PROGRAM F25_CylindersCtrl
VAR
	aCylinderCtrl		:ARRAY[1..cMAX_CYLINDERS] OF  FB_Cylinder;

	bStationHomed		: BOOL;
	bSeqHomingRequest	: BOOL;
	bTestRelease			: BOOL;
END_VAR
VAR // added by the converter: edge detectors and wires of the graphical bodies
    _w1, _w2, _w3, _w4, _w5, _w6, _w7 : BOOL;
END_VAR

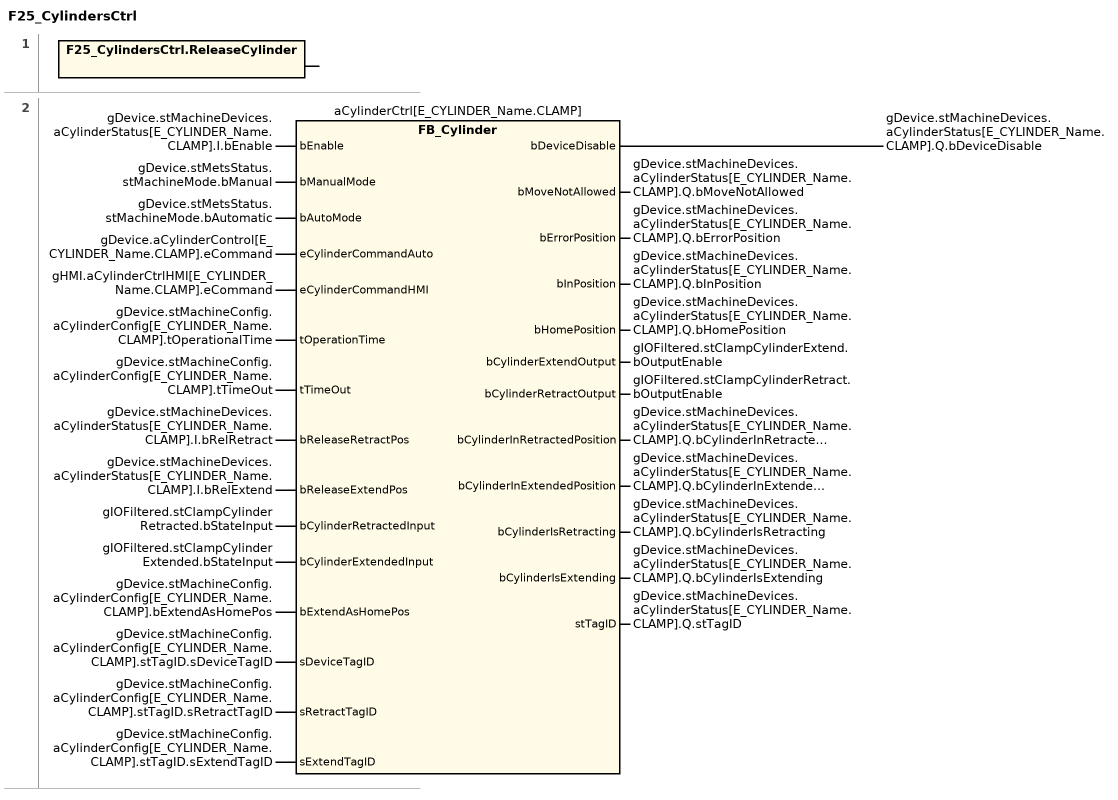
// NETWORK 1
F25_CylindersCtrl.ReleaseCylinder();

// NETWORK 2
aCylinderCtrl[E_CYLINDER_Name.CLAMP](
    bEnable := gDevice.stMachineDevices.aCylinderStatus[E_CYLINDER_Name.CLAMP].I.bEnable,
    bManualMode := gDevice.stMetsStatus.stMachineMode.bManual,
    bAutoMode := gDevice.stMetsStatus.stMachineMode.bAutomatic,
    eCylinderCommandAuto := gDevice.aCylinderControl[E_CYLINDER_Name.CLAMP].eCommand,
    eCylinderCommandHMI := gHMI.aCylinderCtrlHMI[E_CYLINDER_Name.CLAMP].eCommand,
    tOperationTime := gDevice.stMachineConfig.aCylinderConfig[E_CYLINDER_Name.CLAMP].tOperationalTime,
    tTimeOut := gDevice.stMachineConfig.aCylinderConfig[E_CYLINDER_Name.CLAMP].tTimeOut,
    bReleaseRetractPos := gDevice.stMachineDevices.aCylinderStatus[E_CYLINDER_Name.CLAMP].I.bRelRetract,
    bReleaseExtendPos := gDevice.stMachineDevices.aCylinderStatus[E_CYLINDER_Name.CLAMP].I.bRelExtend,
    bCylinderRetractedInput := gIOFiltered.stClampCylinderRetracted.bStateInput,
    bCylinderExtendedInput := gIOFiltered.stClampCylinderExtended.bStateInput,
    bExtendAsHomePos := gDevice.stMachineConfig.aCylinderConfig[E_CYLINDER_Name.CLAMP].bExtendAsHomePos,
    sDeviceTagID := gDevice.stMachineConfig.aCylinderConfig[E_CYLINDER_Name.CLAMP].stTagID.sDeviceTagID,
    sRetractTagID := gDevice.stMachineConfig.aCylinderConfig[E_CYLINDER_Name.CLAMP].stTagID.sRetractTagID,
    sExtendTagID := gDevice.stMachineConfig.aCylinderConfig[E_CYLINDER_Name.CLAMP].stTagID.sExtendTagID,
    bMoveNotAllowed => gDevice.stMachineDevices.aCylinderStatus[E_CYLINDER_Name.CLAMP].Q.bMoveNotAllowed,
    bErrorPosition => gDevice.stMachineDevices.aCylinderStatus[E_CYLINDER_Name.CLAMP].Q.bErrorPosition,
    bInPosition => gDevice.stMachineDevices.aCylinderStatus[E_CYLINDER_Name.CLAMP].Q.bInPosition,
    bHomePosition => gDevice.stMachineDevices.aCylinderStatus[E_CYLINDER_Name.CLAMP].Q.bHomePosition,
    bCylinderExtendOutput => gIOFiltered.stClampCylinderExtend.bOutputEnable,
    bCylinderRetractOutput => gIOFiltered.stClampCylinderRetract.bOutputEnable,
    bCylinderInRetractedPosition => gDevice.stMachineDevices.aCylinderStatus[E_CYLINDER_Name.CLAMP].Q.bCylinderInRetractedPosition,
    bCylinderInExtendedPosition => gDevice.stMachineDevices.aCylinderStatus[E_CYLINDER_Name.CLAMP].Q.bCylinderInExtendedPosition,
    bCylinderIsRetracting => gDevice.stMachineDevices.aCylinderStatus[E_CYLINDER_Name.CLAMP].Q.bCylinderIsRetracting,
    bCylinderIsExtending => gDevice.stMachineDevices.aCylinderStatus[E_CYLINDER_Name.CLAMP].Q.bCylinderIsExtending,
    stTagID => gDevice.stMachineDevices.aCylinderStatus[E_CYLINDER_Name.CLAMP].Q.stTagID); // FB_Cylinder
gDevice.stMachineDevices.aCylinderStatus[E_CYLINDER_Name.CLAMP].Q.bDeviceDisable := aCylinderCtrl[E_CYLINDER_Name.CLAMP].bDeviceDisable;

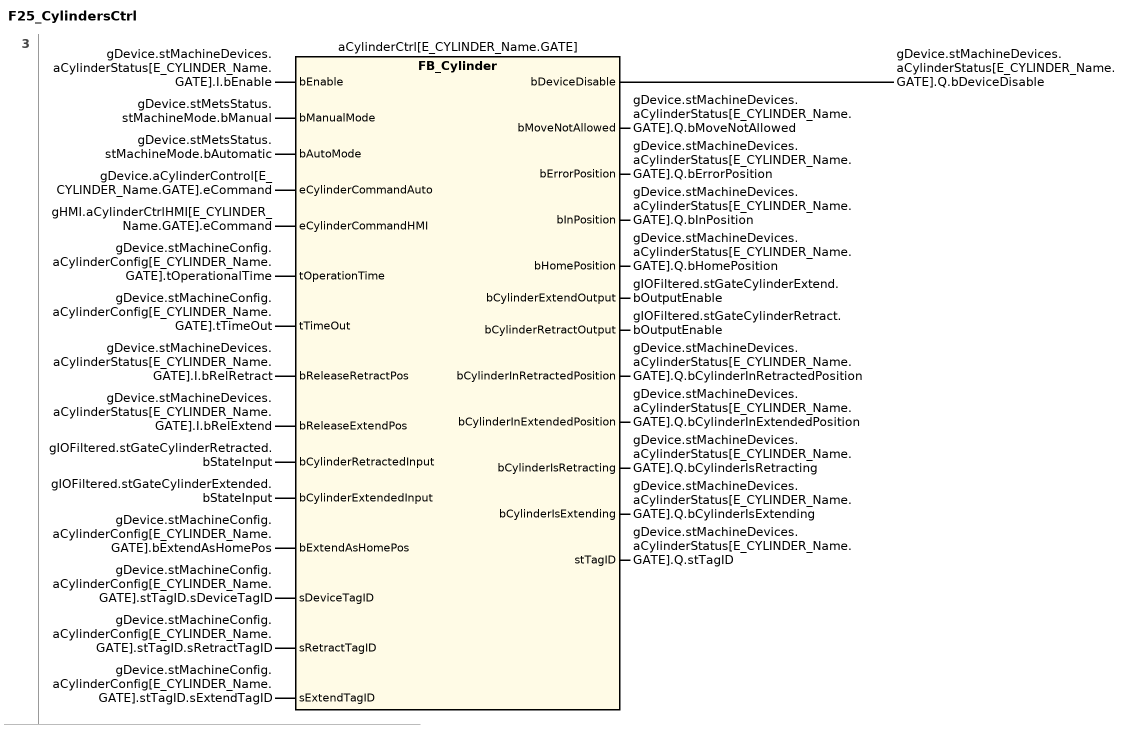
// NETWORK 3
aCylinderCtrl[E_CYLINDER_Name.GATE](
    bEnable := gDevice.stMachineDevices.aCylinderStatus[E_CYLINDER_Name.GATE].I.bEnable,
    bManualMode := gDevice.stMetsStatus.stMachineMode.bManual,
    bAutoMode := gDevice.stMetsStatus.stMachineMode.bAutomatic,
    eCylinderCommandAuto := gDevice.aCylinderControl[E_CYLINDER_Name.GATE].eCommand,
    eCylinderCommandHMI := gHMI.aCylinderCtrlHMI[E_CYLINDER_Name.GATE].eCommand,
    tOperationTime := gDevice.stMachineConfig.aCylinderConfig[E_CYLINDER_Name.GATE].tOperationalTime,
    tTimeOut := gDevice.stMachineConfig.aCylinderConfig[E_CYLINDER_Name.GATE].tTimeOut,
    bReleaseRetractPos := gDevice.stMachineDevices.aCylinderStatus[E_CYLINDER_Name.GATE].I.bRelRetract,
    bReleaseExtendPos := gDevice.stMachineDevices.aCylinderStatus[E_CYLINDER_Name.GATE].I.bRelExtend,
    bCylinderRetractedInput := gIOFiltered.stGateCylinderRetracted.bStateInput,
    bCylinderExtendedInput := gIOFiltered.stGateCylinderExtended.bStateInput,
    bExtendAsHomePos := gDevice.stMachineConfig.aCylinderConfig[E_CYLINDER_Name.GATE].bExtendAsHomePos,
    sDeviceTagID := gDevice.stMachineConfig.aCylinderConfig[E_CYLINDER_Name.GATE].stTagID.sDeviceTagID,
    sRetractTagID := gDevice.stMachineConfig.aCylinderConfig[E_CYLINDER_Name.GATE].stTagID.sRetractTagID,
    sExtendTagID := gDevice.stMachineConfig.aCylinderConfig[E_CYLINDER_Name.GATE].stTagID.sExtendTagID,
    bMoveNotAllowed => gDevice.stMachineDevices.aCylinderStatus[E_CYLINDER_Name.GATE].Q.bMoveNotAllowed,
    bErrorPosition => gDevice.stMachineDevices.aCylinderStatus[E_CYLINDER_Name.GATE].Q.bErrorPosition,
    bInPosition => gDevice.stMachineDevices.aCylinderStatus[E_CYLINDER_Name.GATE].Q.bInPosition,
    bHomePosition => gDevice.stMachineDevices.aCylinderStatus[E_CYLINDER_Name.GATE].Q.bHomePosition,
    bCylinderExtendOutput => gIOFiltered.stGateCylinderExtend.bOutputEnable,
    bCylinderRetractOutput => gIOFiltered.stGateCylinderRetract.bOutputEnable,
    bCylinderInRetractedPosition => gDevice.stMachineDevices.aCylinderStatus[E_CYLINDER_Name.GATE].Q.bCylinderInRetractedPosition,
    bCylinderInExtendedPosition => gDevice.stMachineDevices.aCylinderStatus[E_CYLINDER_Name.GATE].Q.bCylinderInExtendedPosition,
    bCylinderIsRetracting => gDevice.stMachineDevices.aCylinderStatus[E_CYLINDER_Name.GATE].Q.bCylinderIsRetracting,
    bCylinderIsExtending => gDevice.stMachineDevices.aCylinderStatus[E_CYLINDER_Name.GATE].Q.bCylinderIsExtending,
    stTagID => gDevice.stMachineDevices.aCylinderStatus[E_CYLINDER_Name.GATE].Q.stTagID); // FB_Cylinder
gDevice.stMachineDevices.aCylinderStatus[E_CYLINDER_Name.GATE].Q.bDeviceDisable := aCylinderCtrl[E_CYLINDER_Name.GATE].bDeviceDisable;

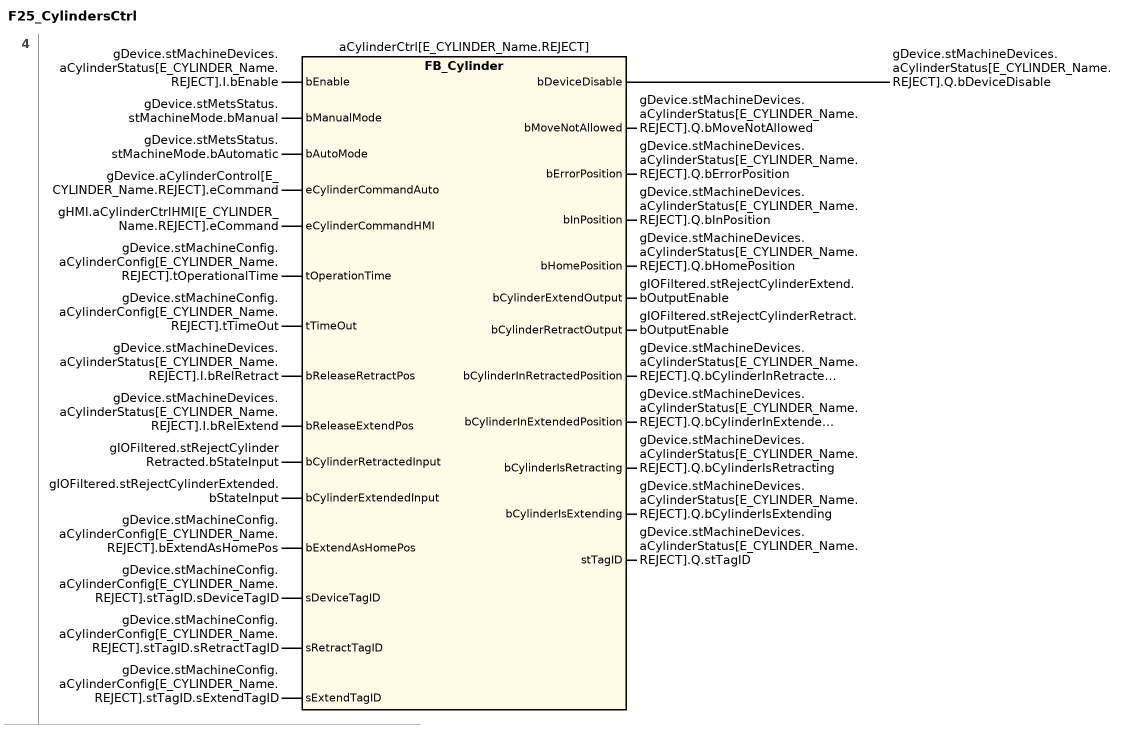
// NETWORK 4
aCylinderCtrl[E_CYLINDER_Name.REJECT](
    bEnable := gDevice.stMachineDevices.aCylinderStatus[E_CYLINDER_Name.REJECT].I.bEnable,
    bManualMode := gDevice.stMetsStatus.stMachineMode.bManual,
    bAutoMode := gDevice.stMetsStatus.stMachineMode.bAutomatic,
    eCylinderCommandAuto := gDevice.aCylinderControl[E_CYLINDER_Name.REJECT].eCommand,
    eCylinderCommandHMI := gHMI.aCylinderCtrlHMI[E_CYLINDER_Name.REJECT].eCommand,
    tOperationTime := gDevice.stMachineConfig.aCylinderConfig[E_CYLINDER_Name.REJECT].tOperationalTime,
    tTimeOut := gDevice.stMachineConfig.aCylinderConfig[E_CYLINDER_Name.REJECT].tTimeOut,
    bReleaseRetractPos := gDevice.stMachineDevices.aCylinderStatus[E_CYLINDER_Name.REJECT].I.bRelRetract,
    bReleaseExtendPos := gDevice.stMachineDevices.aCylinderStatus[E_CYLINDER_Name.REJECT].I.bRelExtend,
    bCylinderRetractedInput := gIOFiltered.stRejectCylinderRetracted.bStateInput,
    bCylinderExtendedInput := gIOFiltered.stRejectCylinderExtended.bStateInput,
    bExtendAsHomePos := gDevice.stMachineConfig.aCylinderConfig[E_CYLINDER_Name.REJECT].bExtendAsHomePos,
    sDeviceTagID := gDevice.stMachineConfig.aCylinderConfig[E_CYLINDER_Name.REJECT].stTagID.sDeviceTagID,
    sRetractTagID := gDevice.stMachineConfig.aCylinderConfig[E_CYLINDER_Name.REJECT].stTagID.sRetractTagID,
    sExtendTagID := gDevice.stMachineConfig.aCylinderConfig[E_CYLINDER_Name.REJECT].stTagID.sExtendTagID,
    bMoveNotAllowed => gDevice.stMachineDevices.aCylinderStatus[E_CYLINDER_Name.REJECT].Q.bMoveNotAllowed,
    bErrorPosition => gDevice.stMachineDevices.aCylinderStatus[E_CYLINDER_Name.REJECT].Q.bErrorPosition,
    bInPosition => gDevice.stMachineDevices.aCylinderStatus[E_CYLINDER_Name.REJECT].Q.bInPosition,
    bHomePosition => gDevice.stMachineDevices.aCylinderStatus[E_CYLINDER_Name.REJECT].Q.bHomePosition,
    bCylinderExtendOutput => gIOFiltered.stRejectCylinderExtend.bOutputEnable,
    bCylinderRetractOutput => gIOFiltered.stRejectCylinderRetract.bOutputEnable,
    bCylinderInRetractedPosition => gDevice.stMachineDevices.aCylinderStatus[E_CYLINDER_Name.REJECT].Q.bCylinderInRetractedPosition,
    bCylinderInExtendedPosition => gDevice.stMachineDevices.aCylinderStatus[E_CYLINDER_Name.REJECT].Q.bCylinderInExtendedPosition,
    bCylinderIsRetracting => gDevice.stMachineDevices.aCylinderStatus[E_CYLINDER_Name.REJECT].Q.bCylinderIsRetracting,
    bCylinderIsExtending => gDevice.stMachineDevices.aCylinderStatus[E_CYLINDER_Name.REJECT].Q.bCylinderIsExtending,
    stTagID => gDevice.stMachineDevices.aCylinderStatus[E_CYLINDER_Name.REJECT].Q.stTagID); // FB_Cylinder
gDevice.stMachineDevices.aCylinderStatus[E_CYLINDER_Name.REJECT].Q.bDeviceDisable := aCylinderCtrl[E_CYLINDER_Name.REJECT].bDeviceDisable;

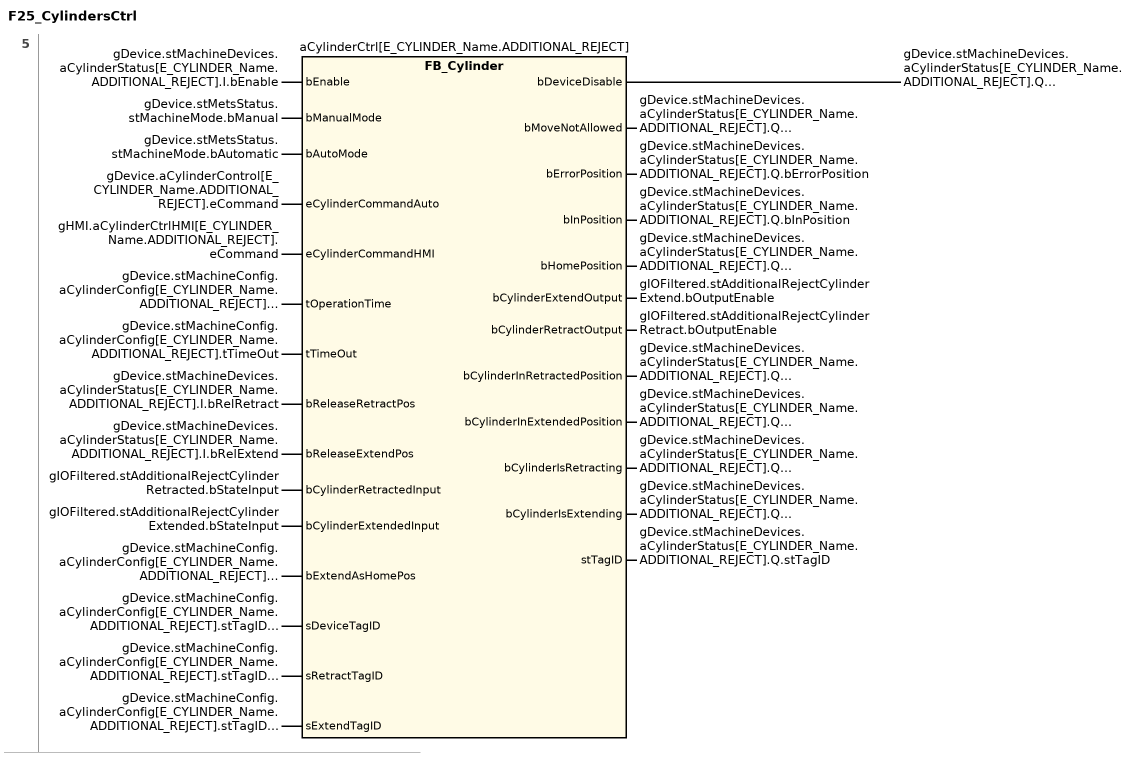
// NETWORK 5
aCylinderCtrl[E_CYLINDER_Name.ADDITIONAL_REJECT](
    bEnable := gDevice.stMachineDevices.aCylinderStatus[E_CYLINDER_Name.ADDITIONAL_REJECT].I.bEnable,
    bManualMode := gDevice.stMetsStatus.stMachineMode.bManual,
    bAutoMode := gDevice.stMetsStatus.stMachineMode.bAutomatic,
    eCylinderCommandAuto := gDevice.aCylinderControl[E_CYLINDER_Name.ADDITIONAL_REJECT].eCommand,
    eCylinderCommandHMI := gHMI.aCylinderCtrlHMI[E_CYLINDER_Name.ADDITIONAL_REJECT].eCommand,
    tOperationTime := gDevice.stMachineConfig.aCylinderConfig[E_CYLINDER_Name.ADDITIONAL_REJECT].tOperationalTime,
    tTimeOut := gDevice.stMachineConfig.aCylinderConfig[E_CYLINDER_Name.ADDITIONAL_REJECT].tTimeOut,
    bReleaseRetractPos := gDevice.stMachineDevices.aCylinderStatus[E_CYLINDER_Name.ADDITIONAL_REJECT].I.bRelRetract,
    bReleaseExtendPos := gDevice.stMachineDevices.aCylinderStatus[E_CYLINDER_Name.ADDITIONAL_REJECT].I.bRelExtend,
    bCylinderRetractedInput := gIOFiltered.stAdditionalRejectCylinderRetracted.bStateInput,
    bCylinderExtendedInput := gIOFiltered.stAdditionalRejectCylinderExtended.bStateInput,
    bExtendAsHomePos := gDevice.stMachineConfig.aCylinderConfig[E_CYLINDER_Name.ADDITIONAL_REJECT].bExtendAsHomePos,
    sDeviceTagID := gDevice.stMachineConfig.aCylinderConfig[E_CYLINDER_Name.ADDITIONAL_REJECT].stTagID.sDeviceTagID,
    sRetractTagID := gDevice.stMachineConfig.aCylinderConfig[E_CYLINDER_Name.ADDITIONAL_REJECT].stTagID.sRetractTagID,
    sExtendTagID := gDevice.stMachineConfig.aCylinderConfig[E_CYLINDER_Name.ADDITIONAL_REJECT].stTagID.sExtendTagID,
    bMoveNotAllowed => gDevice.stMachineDevices.aCylinderStatus[E_CYLINDER_Name.ADDITIONAL_REJECT].Q.bMoveNotAllowed,
    bErrorPosition => gDevice.stMachineDevices.aCylinderStatus[E_CYLINDER_Name.ADDITIONAL_REJECT].Q.bErrorPosition,
    bInPosition => gDevice.stMachineDevices.aCylinderStatus[E_CYLINDER_Name.ADDITIONAL_REJECT].Q.bInPosition,
    bHomePosition => gDevice.stMachineDevices.aCylinderStatus[E_CYLINDER_Name.ADDITIONAL_REJECT].Q.bHomePosition,
    bCylinderExtendOutput => gIOFiltered.stAdditionalRejectCylinderExtend.bOutputEnable,
    bCylinderRetractOutput => gIOFiltered.stAdditionalRejectCylinderRetract.bOutputEnable,
    bCylinderInRetractedPosition => gDevice.stMachineDevices.aCylinderStatus[E_CYLINDER_Name.ADDITIONAL_REJECT].Q.bCylinderInRetractedPosition,
    bCylinderInExtendedPosition => gDevice.stMachineDevices.aCylinderStatus[E_CYLINDER_Name.ADDITIONAL_REJECT].Q.bCylinderInExtendedPosition,
    bCylinderIsRetracting => gDevice.stMachineDevices.aCylinderStatus[E_CYLINDER_Name.ADDITIONAL_REJECT].Q.bCylinderIsRetracting,
    bCylinderIsExtending => gDevice.stMachineDevices.aCylinderStatus[E_CYLINDER_Name.ADDITIONAL_REJECT].Q.bCylinderIsExtending,
    stTagID => gDevice.stMachineDevices.aCylinderStatus[E_CYLINDER_Name.ADDITIONAL_REJECT].Q.stTagID); // FB_Cylinder
gDevice.stMachineDevices.aCylinderStatus[E_CYLINDER_Name.ADDITIONAL_REJECT].Q.bDeviceDisable := aCylinderCtrl[E_CYLINDER_Name.ADDITIONAL_REJECT].bDeviceDisable;

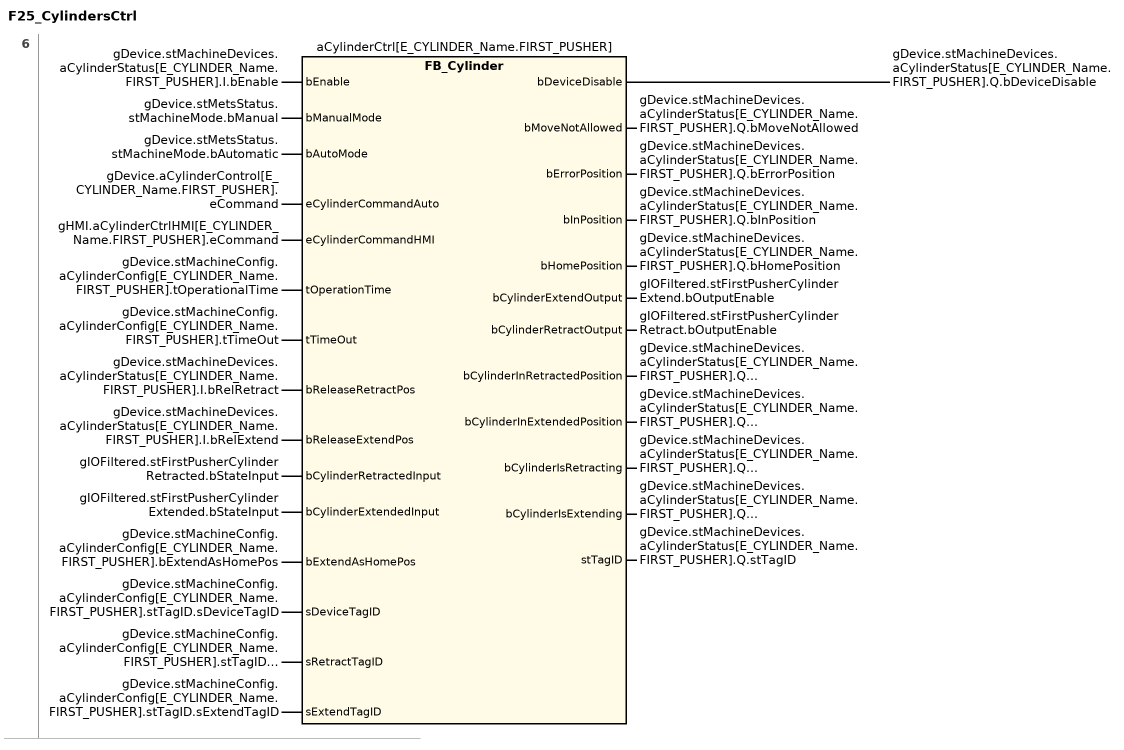
// NETWORK 6
aCylinderCtrl[E_CYLINDER_Name.FIRST_PUSHER](
    bEnable := gDevice.stMachineDevices.aCylinderStatus[E_CYLINDER_Name.FIRST_PUSHER].I.bEnable,
    bManualMode := gDevice.stMetsStatus.stMachineMode.bManual,
    bAutoMode := gDevice.stMetsStatus.stMachineMode.bAutomatic,
    eCylinderCommandAuto := gDevice.aCylinderControl[E_CYLINDER_Name.FIRST_PUSHER].eCommand,
    eCylinderCommandHMI := gHMI.aCylinderCtrlHMI[E_CYLINDER_Name.FIRST_PUSHER].eCommand,
    tOperationTime := gDevice.stMachineConfig.aCylinderConfig[E_CYLINDER_Name.FIRST_PUSHER].tOperationalTime,
    tTimeOut := gDevice.stMachineConfig.aCylinderConfig[E_CYLINDER_Name.FIRST_PUSHER].tTimeOut,
    bReleaseRetractPos := gDevice.stMachineDevices.aCylinderStatus[E_CYLINDER_Name.FIRST_PUSHER].I.bRelRetract,
    bReleaseExtendPos := gDevice.stMachineDevices.aCylinderStatus[E_CYLINDER_Name.FIRST_PUSHER].I.bRelExtend,
    bCylinderRetractedInput := gIOFiltered.stFirstPusherCylinderRetracted.bStateInput,
    bCylinderExtendedInput := gIOFiltered.stFirstPusherCylinderExtended.bStateInput,
    bExtendAsHomePos := gDevice.stMachineConfig.aCylinderConfig[E_CYLINDER_Name.FIRST_PUSHER].bExtendAsHomePos,
    sDeviceTagID := gDevice.stMachineConfig.aCylinderConfig[E_CYLINDER_Name.FIRST_PUSHER].stTagID.sDeviceTagID,
    sRetractTagID := gDevice.stMachineConfig.aCylinderConfig[E_CYLINDER_Name.FIRST_PUSHER].stTagID.sRetractTagID,
    sExtendTagID := gDevice.stMachineConfig.aCylinderConfig[E_CYLINDER_Name.FIRST_PUSHER].stTagID.sExtendTagID,
    bMoveNotAllowed => gDevice.stMachineDevices.aCylinderStatus[E_CYLINDER_Name.FIRST_PUSHER].Q.bMoveNotAllowed,
    bErrorPosition => gDevice.stMachineDevices.aCylinderStatus[E_CYLINDER_Name.FIRST_PUSHER].Q.bErrorPosition,
    bInPosition => gDevice.stMachineDevices.aCylinderStatus[E_CYLINDER_Name.FIRST_PUSHER].Q.bInPosition,
    bHomePosition => gDevice.stMachineDevices.aCylinderStatus[E_CYLINDER_Name.FIRST_PUSHER].Q.bHomePosition,
    bCylinderExtendOutput => gIOFiltered.stFirstPusherCylinderExtend.bOutputEnable,
    bCylinderRetractOutput => gIOFiltered.stFirstPusherCylinderRetract.bOutputEnable,
    bCylinderInRetractedPosition => gDevice.stMachineDevices.aCylinderStatus[E_CYLINDER_Name.FIRST_PUSHER].Q.bCylinderInRetractedPosition,
    bCylinderInExtendedPosition => gDevice.stMachineDevices.aCylinderStatus[E_CYLINDER_Name.FIRST_PUSHER].Q.bCylinderInExtendedPosition,
    bCylinderIsRetracting => gDevice.stMachineDevices.aCylinderStatus[E_CYLINDER_Name.FIRST_PUSHER].Q.bCylinderIsRetracting,
    bCylinderIsExtending => gDevice.stMachineDevices.aCylinderStatus[E_CYLINDER_Name.FIRST_PUSHER].Q.bCylinderIsExtending,
    stTagID => gDevice.stMachineDevices.aCylinderStatus[E_CYLINDER_Name.FIRST_PUSHER].Q.stTagID); // FB_Cylinder
gDevice.stMachineDevices.aCylinderStatus[E_CYLINDER_Name.FIRST_PUSHER].Q.bDeviceDisable := aCylinderCtrl[E_CYLINDER_Name.FIRST_PUSHER].bDeviceDisable;

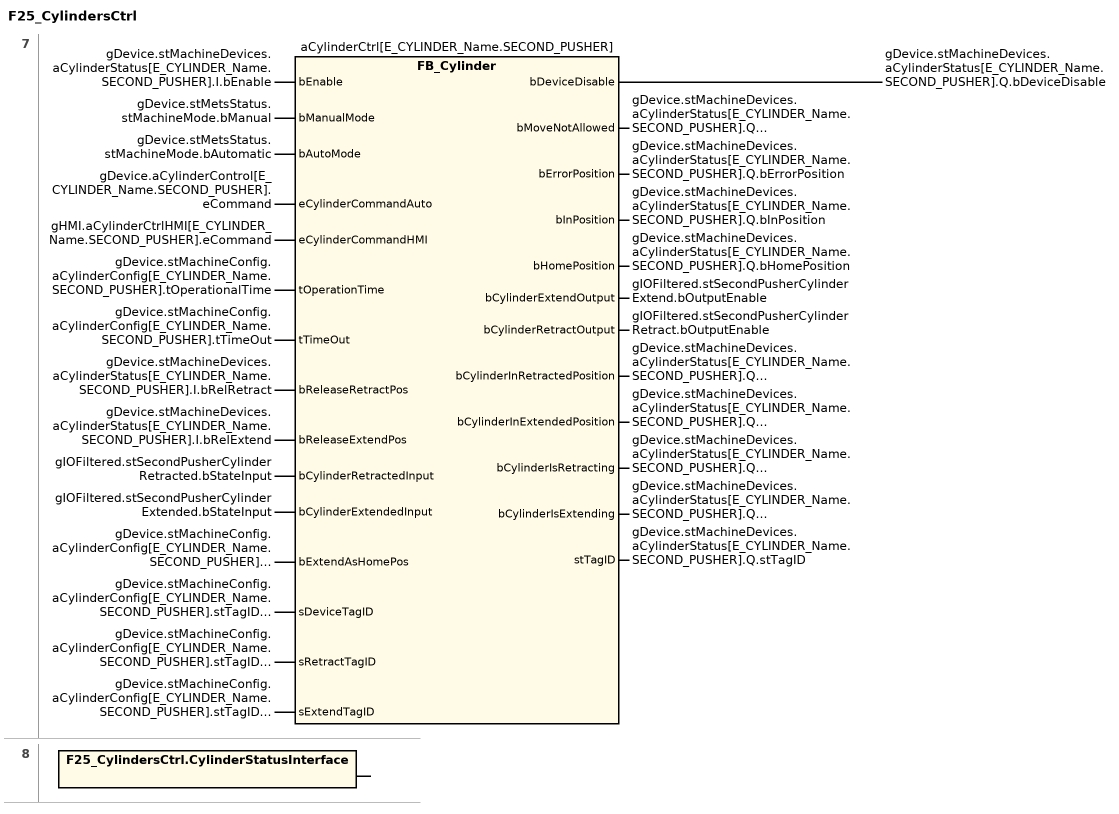
// NETWORK 7
aCylinderCtrl[E_CYLINDER_Name.SECOND_PUSHER](
    bEnable := gDevice.stMachineDevices.aCylinderStatus[E_CYLINDER_Name.SECOND_PUSHER].I.bEnable,
    bManualMode := gDevice.stMetsStatus.stMachineMode.bManual,
    bAutoMode := gDevice.stMetsStatus.stMachineMode.bAutomatic,
    eCylinderCommandAuto := gDevice.aCylinderControl[E_CYLINDER_Name.SECOND_PUSHER].eCommand,
    eCylinderCommandHMI := gHMI.aCylinderCtrlHMI[E_CYLINDER_Name.SECOND_PUSHER].eCommand,
    tOperationTime := gDevice.stMachineConfig.aCylinderConfig[E_CYLINDER_Name.SECOND_PUSHER].tOperationalTime,
    tTimeOut := gDevice.stMachineConfig.aCylinderConfig[E_CYLINDER_Name.SECOND_PUSHER].tTimeOut,
    bReleaseRetractPos := gDevice.stMachineDevices.aCylinderStatus[E_CYLINDER_Name.SECOND_PUSHER].I.bRelRetract,
    bReleaseExtendPos := gDevice.stMachineDevices.aCylinderStatus[E_CYLINDER_Name.SECOND_PUSHER].I.bRelExtend,
    bCylinderRetractedInput := gIOFiltered.stSecondPusherCylinderRetracted.bStateInput,
    bCylinderExtendedInput := gIOFiltered.stSecondPusherCylinderExtended.bStateInput,
    bExtendAsHomePos := gDevice.stMachineConfig.aCylinderConfig[E_CYLINDER_Name.SECOND_PUSHER].bExtendAsHomePos,
    sDeviceTagID := gDevice.stMachineConfig.aCylinderConfig[E_CYLINDER_Name.SECOND_PUSHER].stTagID.sDeviceTagID,
    sRetractTagID := gDevice.stMachineConfig.aCylinderConfig[E_CYLINDER_Name.SECOND_PUSHER].stTagID.sRetractTagID,
    sExtendTagID := gDevice.stMachineConfig.aCylinderConfig[E_CYLINDER_Name.SECOND_PUSHER].stTagID.sExtendTagID,
    bMoveNotAllowed => gDevice.stMachineDevices.aCylinderStatus[E_CYLINDER_Name.SECOND_PUSHER].Q.bMoveNotAllowed,
    bErrorPosition => gDevice.stMachineDevices.aCylinderStatus[E_CYLINDER_Name.SECOND_PUSHER].Q.bErrorPosition,
    bInPosition => gDevice.stMachineDevices.aCylinderStatus[E_CYLINDER_Name.SECOND_PUSHER].Q.bInPosition,
    bHomePosition => gDevice.stMachineDevices.aCylinderStatus[E_CYLINDER_Name.SECOND_PUSHER].Q.bHomePosition,
    bCylinderExtendOutput => gIOFiltered.stSecondPusherCylinderExtend.bOutputEnable,
    bCylinderRetractOutput => gIOFiltered.stSecondPusherCylinderRetract.bOutputEnable,
    bCylinderInRetractedPosition => gDevice.stMachineDevices.aCylinderStatus[E_CYLINDER_Name.SECOND_PUSHER].Q.bCylinderInRetractedPosition,
    bCylinderInExtendedPosition => gDevice.stMachineDevices.aCylinderStatus[E_CYLINDER_Name.SECOND_PUSHER].Q.bCylinderInExtendedPosition,
    bCylinderIsRetracting => gDevice.stMachineDevices.aCylinderStatus[E_CYLINDER_Name.SECOND_PUSHER].Q.bCylinderIsRetracting,
    bCylinderIsExtending => gDevice.stMachineDevices.aCylinderStatus[E_CYLINDER_Name.SECOND_PUSHER].Q.bCylinderIsExtending,
    stTagID => gDevice.stMachineDevices.aCylinderStatus[E_CYLINDER_Name.SECOND_PUSHER].Q.stTagID); // FB_Cylinder
gDevice.stMachineDevices.aCylinderStatus[E_CYLINDER_Name.SECOND_PUSHER].Q.bDeviceDisable := aCylinderCtrl[E_CYLINDER_Name.SECOND_PUSHER].bDeviceDisable;

// NETWORK 8
F25_CylindersCtrl.CylinderStatusInterface();

ACTION CylinderStatusInterface:
MEMMOVE(ADR(gHMI.aCylinderStatusHMI[E_CYLINDER_Name.CLAMP]), ADR(gDevice.stMachineDevices.aCylinderStatus[E_CYLINDER_Name.CLAMP].Q),SIZEOF( gDevice.stMachineDevices.aCylinderStatus[E_CYLINDER_Name.CLAMP].Q));
MEMMOVE(ADR(gHMI.aCylinderStatusHMI[E_CYLINDER_Name.GATE]), ADR(gDevice.stMachineDevices.aCylinderStatus[E_CYLINDER_Name.GATE].Q),SIZEOF( gDevice.stMachineDevices.aCylinderStatus[E_CYLINDER_Name.GATE].Q));
MEMMOVE(ADR(gHMI.aCylinderStatusHMI[E_CYLINDER_Name.REJECT]), ADR(gDevice.stMachineDevices.aCylinderStatus[E_CYLINDER_Name.REJECT].Q),SIZEOF( gDevice.stMachineDevices.aCylinderStatus[E_CYLINDER_Name.REJECT].Q));
MEMMOVE(ADR(gHMI.aCylinderStatusHMI[E_CYLINDER_Name.ADDITIONAL_REJECT]), ADR(gDevice.stMachineDevices.aCylinderStatus[E_CYLINDER_Name.ADDITIONAL_REJECT].Q),SIZEOF( gDevice.stMachineDevices.aCylinderStatus[E_CYLINDER_Name.ADDITIONAL_REJECT].Q));
MEMMOVE(ADR(gHMI.aCylinderStatusHMI[E_CYLINDER_Name.FIRST_PUSHER]), ADR(gDevice.stMachineDevices.aCylinderStatus[E_CYLINDER_Name.FIRST_PUSHER].Q),SIZEOF( gDevice.stMachineDevices.aCylinderStatus[E_CYLINDER_Name.FIRST_PUSHER].Q));
MEMMOVE(ADR(gHMI.aCylinderStatusHMI[E_CYLINDER_Name.SECOND_PUSHER]), ADR(gDevice.stMachineDevices.aCylinderStatus[E_CYLINDER_Name.SECOND_PUSHER].Q),SIZEOF( gDevice.stMachineDevices.aCylinderStatus[E_CYLINDER_Name.SECOND_PUSHER].Q));
END_ACTION

ACTION ReleaseCylinder:
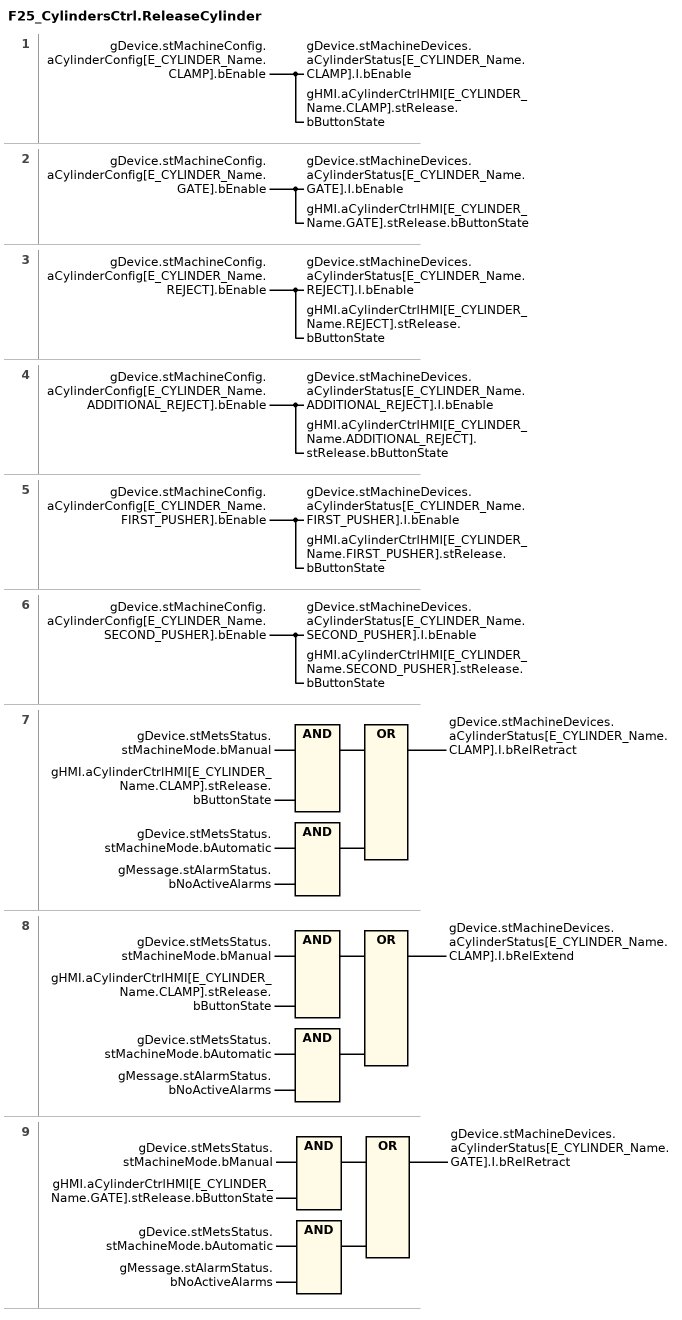
// NETWORK 1
_w1 := gDevice.stMachineConfig.aCylinderConfig[E_CYLINDER_Name.CLAMP].bEnable;
gDevice.stMachineDevices.aCylinderStatus[E_CYLINDER_Name.CLAMP].I.bEnable := _w1;
gHMI.aCylinderCtrlHMI[E_CYLINDER_Name.CLAMP].stRelease.bButtonState := _w1;

// NETWORK 2
_w2 := gDevice.stMachineConfig.aCylinderConfig[E_CYLINDER_Name.GATE].bEnable;
gDevice.stMachineDevices.aCylinderStatus[E_CYLINDER_Name.GATE].I.bEnable := _w2;
gHMI.aCylinderCtrlHMI[E_CYLINDER_Name.GATE].stRelease.bButtonState := _w2;

// NETWORK 3
_w3 := gDevice.stMachineConfig.aCylinderConfig[E_CYLINDER_Name.REJECT].bEnable;
gDevice.stMachineDevices.aCylinderStatus[E_CYLINDER_Name.REJECT].I.bEnable := _w3;
gHMI.aCylinderCtrlHMI[E_CYLINDER_Name.REJECT].stRelease.bButtonState := _w3;

// NETWORK 4
_w4 := gDevice.stMachineConfig.aCylinderConfig[E_CYLINDER_Name.ADDITIONAL_REJECT].bEnable;
gDevice.stMachineDevices.aCylinderStatus[E_CYLINDER_Name.ADDITIONAL_REJECT].I.bEnable := _w4;
gHMI.aCylinderCtrlHMI[E_CYLINDER_Name.ADDITIONAL_REJECT].stRelease.bButtonState := _w4;

// NETWORK 5
_w5 := gDevice.stMachineConfig.aCylinderConfig[E_CYLINDER_Name.FIRST_PUSHER].bEnable;
gDevice.stMachineDevices.aCylinderStatus[E_CYLINDER_Name.FIRST_PUSHER].I.bEnable := _w5;
gHMI.aCylinderCtrlHMI[E_CYLINDER_Name.FIRST_PUSHER].stRelease.bButtonState := _w5;

// NETWORK 6
_w6 := gDevice.stMachineConfig.aCylinderConfig[E_CYLINDER_Name.SECOND_PUSHER].bEnable;
gDevice.stMachineDevices.aCylinderStatus[E_CYLINDER_Name.SECOND_PUSHER].I.bEnable := _w6;
gHMI.aCylinderCtrlHMI[E_CYLINDER_Name.SECOND_PUSHER].stRelease.bButtonState := _w6;

// NETWORK 7
gDevice.stMachineDevices.aCylinderStatus[E_CYLINDER_Name.CLAMP].I.bRelRetract := gDevice.stMetsStatus.stMachineMode.bManual AND gHMI.aCylinderCtrlHMI[E_CYLINDER_Name.CLAMP].stRelease.bButtonState OR gDevice.stMetsStatus.stMachineMode.bAutomatic AND gMessage.stAlarmStatus.bNoActiveAlarms;

// NETWORK 8
gDevice.stMachineDevices.aCylinderStatus[E_CYLINDER_Name.CLAMP].I.bRelExtend := gDevice.stMetsStatus.stMachineMode.bManual AND gHMI.aCylinderCtrlHMI[E_CYLINDER_Name.CLAMP].stRelease.bButtonState OR gDevice.stMetsStatus.stMachineMode.bAutomatic AND gMessage.stAlarmStatus.bNoActiveAlarms;

// NETWORK 9
gDevice.stMachineDevices.aCylinderStatus[E_CYLINDER_Name.GATE].I.bRelRetract := gDevice.stMetsStatus.stMachineMode.bManual AND gHMI.aCylinderCtrlHMI[E_CYLINDER_Name.GATE].stRelease.bButtonState OR gDevice.stMetsStatus.stMachineMode.bAutomatic AND gMessage.stAlarmStatus.bNoActiveAlarms;

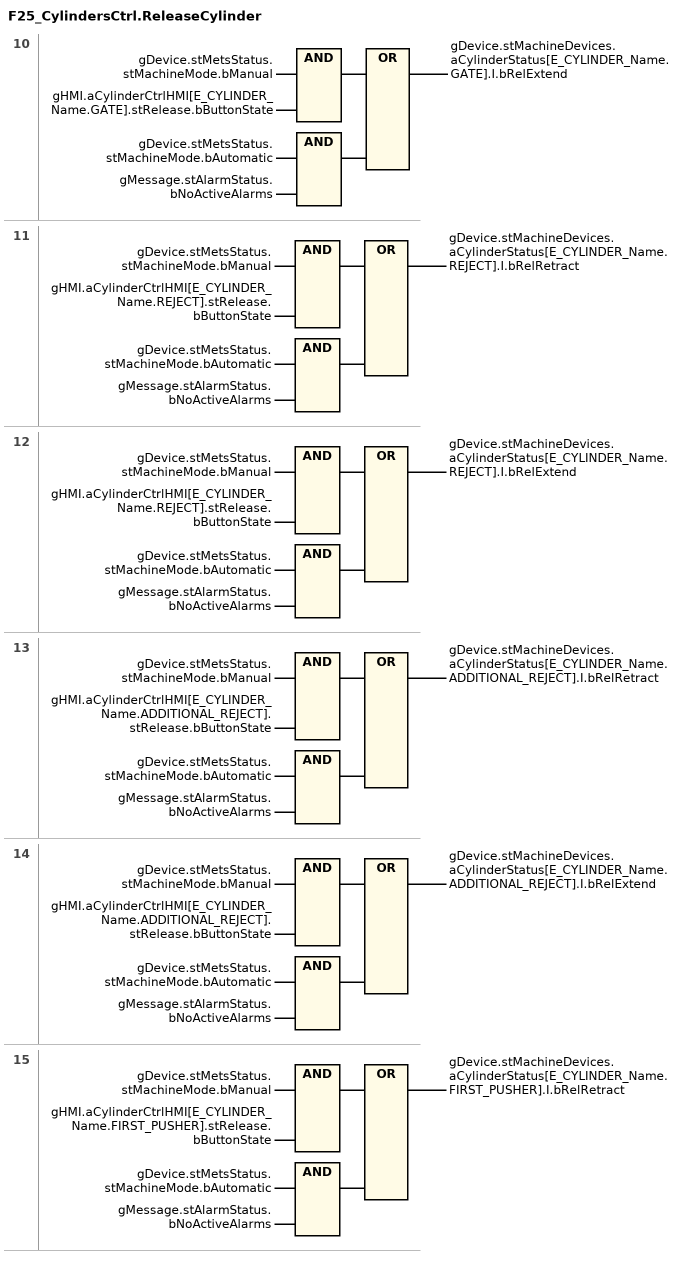
// NETWORK 10
gDevice.stMachineDevices.aCylinderStatus[E_CYLINDER_Name.GATE].I.bRelExtend := gDevice.stMetsStatus.stMachineMode.bManual AND gHMI.aCylinderCtrlHMI[E_CYLINDER_Name.GATE].stRelease.bButtonState OR gDevice.stMetsStatus.stMachineMode.bAutomatic AND gMessage.stAlarmStatus.bNoActiveAlarms;

// NETWORK 11
gDevice.stMachineDevices.aCylinderStatus[E_CYLINDER_Name.REJECT].I.bRelRetract := gDevice.stMetsStatus.stMachineMode.bManual AND gHMI.aCylinderCtrlHMI[E_CYLINDER_Name.REJECT].stRelease.bButtonState OR gDevice.stMetsStatus.stMachineMode.bAutomatic AND gMessage.stAlarmStatus.bNoActiveAlarms;

// NETWORK 12
gDevice.stMachineDevices.aCylinderStatus[E_CYLINDER_Name.REJECT].I.bRelExtend := gDevice.stMetsStatus.stMachineMode.bManual AND gHMI.aCylinderCtrlHMI[E_CYLINDER_Name.REJECT].stRelease.bButtonState OR gDevice.stMetsStatus.stMachineMode.bAutomatic AND gMessage.stAlarmStatus.bNoActiveAlarms;

// NETWORK 13
gDevice.stMachineDevices.aCylinderStatus[E_CYLINDER_Name.ADDITIONAL_REJECT].I.bRelRetract := gDevice.stMetsStatus.stMachineMode.bManual AND gHMI.aCylinderCtrlHMI[E_CYLINDER_Name.ADDITIONAL_REJECT].stRelease.bButtonState OR gDevice.stMetsStatus.stMachineMode.bAutomatic AND gMessage.stAlarmStatus.bNoActiveAlarms;

// NETWORK 14
gDevice.stMachineDevices.aCylinderStatus[E_CYLINDER_Name.ADDITIONAL_REJECT].I.bRelExtend := gDevice.stMetsStatus.stMachineMode.bManual AND gHMI.aCylinderCtrlHMI[E_CYLINDER_Name.ADDITIONAL_REJECT].stRelease.bButtonState OR gDevice.stMetsStatus.stMachineMode.bAutomatic AND gMessage.stAlarmStatus.bNoActiveAlarms;

// NETWORK 15
gDevice.stMachineDevices.aCylinderStatus[E_CYLINDER_Name.FIRST_PUSHER].I.bRelRetract := gDevice.stMetsStatus.stMachineMode.bManual AND gHMI.aCylinderCtrlHMI[E_CYLINDER_Name.FIRST_PUSHER].stRelease.bButtonState OR gDevice.stMetsStatus.stMachineMode.bAutomatic AND gMessage.stAlarmStatus.bNoActiveAlarms;

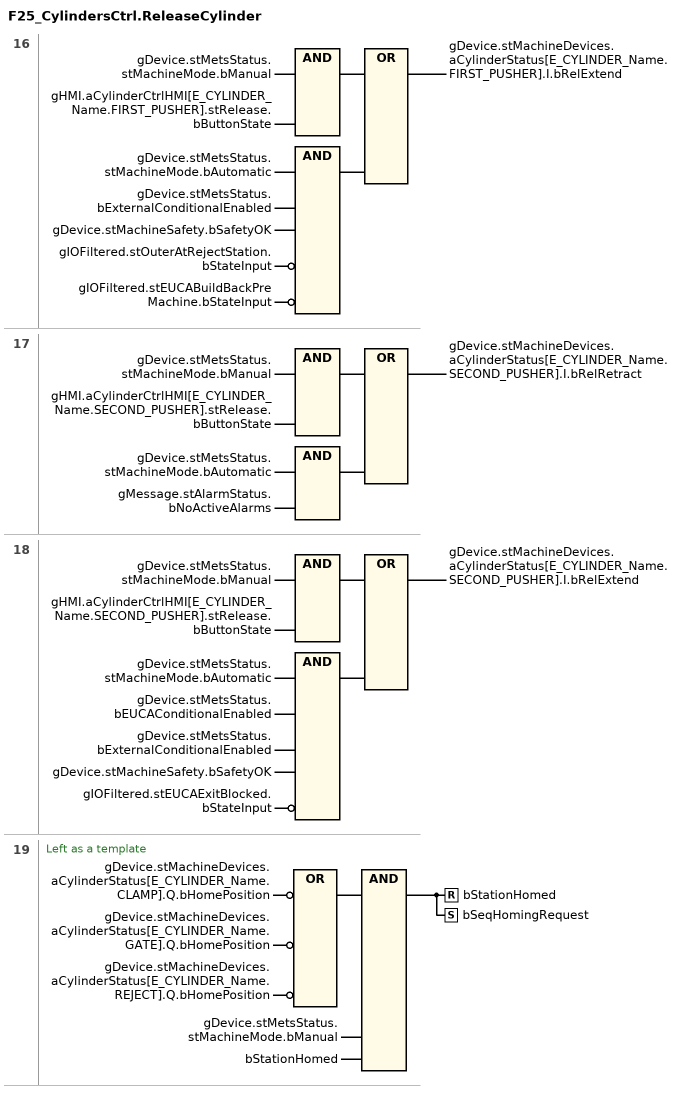
// NETWORK 16
gDevice.stMachineDevices.aCylinderStatus[E_CYLINDER_Name.FIRST_PUSHER].I.bRelExtend := gDevice.stMetsStatus.stMachineMode.bManual AND gHMI.aCylinderCtrlHMI[E_CYLINDER_Name.FIRST_PUSHER].stRelease.bButtonState OR gDevice.stMetsStatus.stMachineMode.bAutomatic AND gDevice.stMetsStatus.bExternalConditionalEnabled AND gDevice.stMachineSafety.bSafetyOK AND NOT gIOFiltered.stOuterAtRejectStation.bStateInput AND NOT gIOFiltered.stEUCABuildBackPreMachine.bStateInput;

// NETWORK 17
gDevice.stMachineDevices.aCylinderStatus[E_CYLINDER_Name.SECOND_PUSHER].I.bRelRetract := gDevice.stMetsStatus.stMachineMode.bManual AND gHMI.aCylinderCtrlHMI[E_CYLINDER_Name.SECOND_PUSHER].stRelease.bButtonState OR gDevice.stMetsStatus.stMachineMode.bAutomatic AND gMessage.stAlarmStatus.bNoActiveAlarms;

// NETWORK 18
gDevice.stMachineDevices.aCylinderStatus[E_CYLINDER_Name.SECOND_PUSHER].I.bRelExtend := gDevice.stMetsStatus.stMachineMode.bManual AND gHMI.aCylinderCtrlHMI[E_CYLINDER_Name.SECOND_PUSHER].stRelease.bButtonState OR gDevice.stMetsStatus.stMachineMode.bAutomatic AND gDevice.stMetsStatus.bEUCAConditionalEnabled AND gDevice.stMetsStatus.bExternalConditionalEnabled AND gDevice.stMachineSafety.bSafetyOK AND NOT gIOFiltered.stEUCAExitBlocked.bStateInput;

// NETWORK 19
// Left as a template
_w7 := (NOT gDevice.stMachineDevices.aCylinderStatus[E_CYLINDER_Name.CLAMP].Q.bHomePosition OR NOT gDevice.stMachineDevices.aCylinderStatus[E_CYLINDER_Name.GATE].Q.bHomePosition OR NOT gDevice.stMachineDevices.aCylinderStatus[E_CYLINDER_Name.REJECT].Q.bHomePosition) AND gDevice.stMetsStatus.stMachineMode.bManual AND bStationHomed;
bStationHomed R= _w7;
bSeqHomingRequest S= _w7;
END_ACTION

END_PROGRAM

(* stored: Version 1.1.0.1
   POU F25_CylindersCtrl: Id {cc3f0596-48ee-4dde-a8ff-21a7772ef767}, SpecialFunc None
   Action CylinderStatusInterface: Id {e0ac35d8-ff3c-47b7-bc4a-cc334808ac9f}
   Action ReleaseCylinder: Id {b7e95581-f4e9-43ed-93a5-ca3939c722bf} *)
